// TIA Portal V17 export
// export: Created 2025-03-10T12:14:37.5345526Z, ExportSetting WithDefaults, DisplayName Totally Integrated Automation Portal, DisplayVersion V17 Update 8, DisplayName TIA Portal Openness, DisplayVersion V17 Update 8, DisplayName TIA Portal Version Control Interface, DisplayVersion V17, DisplayName SINAMICS Startdrive Advanced, DisplayVersion V17 SP2, DisplayName SINAMICS Startdrive G110M, G120, G120C, G120D, G120P, G115D, DisplayVersion V17 SP2, DisplayName SINAMICS Startdrive G130, G150, S120, S150, SINAMICS MV, S210, DisplayVersion V17 SP2, DisplayName STEP 7 Professional, DisplayVersion V17 Update 8, DisplayName SINUMERIK ONE STEP 7 Toolbox, DisplayVersion V17 Update 12, DisplayName SINUMERIK 840D sl STEP 7 Toolbox, DisplayVersion V17 Update 12, DisplayName STEP 7 Safety, DisplayVersion V17 Update 6, DisplayName WinCC Advanced, DisplayVersion V17 Update 8
DATA_BLOCK "LBP_SentronPac"   // DB1001
TITLE = for migration: SENTRON PAC / Para migración: SENTRON PAC / für Migration: SENTRON PAC
{ S7_Optimized_Access := 'FALSE'; DB_Accessible_From_OPC_UA := 'FALSE' }
AUTHOR : SINUMERIK
FAMILY : SINUMERIK_ONE
VERSION : 6.15
// for migration: Interface between user program and operating software, contains signals for SENTRON PAC energy monitoring devices / Para migración: interfaz entre programa de usuario y software operativo, contiene señales para dispositivos de control de la energía SENTRON PAC / für Migration: Schnittstelle zwischen Anwenderprogramm und Betriebssoftware, enthält Signale für SENTRON PAC Energieüberwachungsgeräte
// stored: AutoNumber false, DBAccessibleFromOPCUA false, DBAccessibleFromWebserver true, IsOnlyStoredInLoadMemory false, IsWriteProtectedInAS false
   VAR RETAIN
      ManualVal : Bool;   // Anzeige des manuellen Werts / Display of manual value / Indicación del valor manual
      SentronPacMach : Bool;   // Sentron PAC dargestellte Maschine / Sentron PAC represented machine / Máquina representada en Sentron PAC
      FeedInEnergyReadSP : Bool;   // Zugeführte Energie wird von Sentron PAC gelesen / Feed-in energy read from Sentron PAC / La energía suministrada es leída por Sentron PAC
      FeedBackEnergyReadSP : Bool;   // Rückgespeiste Energie wird von Sentron PAC gelesen / Feed back energy read from Sentron PAC / La energía realimentada es leída por Sentron PAC
      FeedInEnergyReadAuxil : Bool;   // Zugeführte Energie, AUX lesen / Feed-in energy read auxiliary / Energía suministrada, leer AUX
      FeedBackEnergyReadAuxil : Bool;   // Rückgespeiste Energie, AUX lesen / Feed back energy read auxiliary / Energía realimentada, leer AUX
      res0_6 : Bool;   // Reserviert / Reserved / Reservado
      res0_7 : Bool;   // Reserviert / Reserved / Reservado
      MeasAuto : Bool;   // Messung durch PLC-Grundprogramm / Measurement by PLC basic program / Medición por programa básico del PLC
      res1_1 : Bool;   // Reserviert / Reserved / Reservado
      res1_2 : Bool;   // Reserviert / Reserved / Reservado
      res1_3 : Bool;   // Reserviert / Reserved / Reservado
      res1_4 : Bool;   // Reserviert / Reserved / Reservado
      res1_5 : Bool;   // Reserviert / Reserved / Reservado
      res1_6 : Bool;   // Reserviert / Reserved / Reservado
      res1_7 : Bool;   // Reserviert / Reserved / Reservado
      MeasAct : Bool;   // Aktive Messung
      res2_1 : Bool;   // Reserviert / Reserved / Reservado
      res2_2 : Bool;   // Reserviert / Reserved / Reservado
      res2_3 : Bool;   // Reserviert / Reserved / Reservado
      res2_4 : Bool;   // Reserviert / Reserved / Reservado
      res2_5 : Bool;   // Reserviert / Reserved / Reservado
      res2_6 : Bool;   // Reserviert / Reserved / Reservado
      res2_7 : Bool;   // Reserviert / Reserved / Reservado
      EStateOn : Bool;   // Energiezustand Ein / Energy state on / Estado energía Con
      res3_1 : Bool;   // Reserviert / Reserved / Reservado
      res3_2 : Bool;   // Reserviert / Reserved / Reservado
      res3_3 : Bool;   // Reserviert / Reserved / Reservado
      res3_4 : Bool;   // Reserviert / Reserved / Reservado
      res3_5 : Bool;   // Reserviert / Reserved / Reservado
      res3_6 : Bool;   // Reserviert / Reserved / Reservado
      res3_7 : Bool;   // Reserviert / Reserved / Reservado
      ManualValue : Real;   // Manueller Wert / Manual value / Valor manual
      ActivePowerItem : Real;   // Wirkleistung Position / Active power item / Potencia activa, posición
      ActiveEnergyItem : Real;   // Wirkenergie Position / Active energy item / Energía activa, posición
      ReactiveEnergyItem : Real;   // Blindenergie Position / Reactive energy item / Energía reactiva, posición
      ActivePowerSentron : Real;   // Wirkleistung von Sentron / Active power from Sentron / Potencia activa de Sentron
      ActiveEnergySentron : Real;   // Wirkenergie von Sentron / Active energy from Sentron / Energía activa de Sentron
      ReactiveEnergySentron : Real;   // Blindenergie von Sentron / Reactive energy from Sentron / Energía reactiva de Sentron
      ActiveEnergyDay : Real;   // Wirkenergie Tag / Active energy day / Energía activa, día
      ReactiveEnergyDay : Real;   // Blindenergie Tag / Reactive energy day / Energía reactiva, día
      ActiveEnergyPrevDay : Real;   // Wirkenergie Vortag / Active energy previous day / Energía activa, día anterior
      ReactiveEnergyPrevDay : Real;   // Blindenergie Vortag / Reactive energy previous day / Energía reactiva, día anterior
      ActiveEnergyMonth : Real;   // Wirkenergie Monat / Active energy month / Energía activa, mes
      ReactiveEnergyMonth : Real;   // Blindenergie Monat / Reactive energy month / Energía reactiva, mes
      ActiveEnergyPrevMonth : Real;   // Wirkenergie Vormonat / Active energy previous month / Energía activa, mes anterior
      ReactiveEnergyPrevMonth : Real;   // Blindenergie Vormonat / Reactive energy previous month / Energía reactiva, mes anterior
      ActiveEnergyYear : Real;   // Wirkenergie Jahr / Active energy year / Energía activa, año
      ReactiveEnergyYear : Real;   // Blindenergie Jahr / Reactive energy year / Energía reactiva, año
      ActiveEnergyPrevYear : Real;   // Wirkenergie Vorjahr / Active energy previous year / Energía activa, año anterior
      ReactiveEnergyPrevYear : Real;   // Blindenergie Vorjahr / Reactive energy previous year / Energía reactiva, año anterior
      res80 : Byte;   // Reserviert / Reserved / Reservado
      res81 : Byte;   // Reserviert / Reserved / Reservado
      res82 : Byte;   // Reserviert / Reserved / Reservado
      res83 : Byte;   // Reserviert / Reserved / Reservado
      res84 : Byte;   // Reserviert / Reserved / Reservado
      res85 : Byte;   // Reserviert / Reserved / Reservado
      res86 : Byte;   // Reserviert / Reserved / Reservado
      res87 : Byte;   // Reserviert / Reserved / Reservado
      res88 : Real;   // Reserviert / Reserved / Reservado
      res92 : Real;   // Reserviert / Reserved / Reservado
      ProductionAct : Byte;
      ErrDBD20_NAN : Bool;   // DBD20: ungültig (keine Nummer) / DBD20: invalid (not a number) / DBD20: no válido (no es número)
      ErrDBD24_NAN : Bool;   // DBD24: ungültig (keine Nummer) / DBD24: invalid (not a number) / DBD24: no válido (no es número)
      ErrDBD28_NAN : Bool;   // DBD28: ungültig (keine Nummer) / DBD28: invalid (not a number) / DBD28: no válido (no es número)
      res97_3 : Bool;   // Reserviert / Reserved / Reservado
      res97_4 : Bool;   // Reserviert / Reserved / Reservado
      res97_5 : Bool;   // Reserviert / Reserved / Reservado
      res97_6 : Bool;   // Reserviert / Reserved / Reservado
      res97_7 : Bool;   // Reserviert / Reserved / Reservado
      ErrDBD104_NAN : Bool;   // DBD104: ungültig (keine Nummer) / DBD104: invalid (not a number) / DBD104: no válido (no es número)
      ErrDBD144_NAN : Bool;   // DBD144: ungültig (keine Nummer) / DBD144: invalid (not a number) / DBD144: no válido (no es número)
      ErrDBD184_NAN : Bool;   // DBD184: ungültig (keine Nummer) / DBD184: invalid (not a number) / DBD184: no válido (no es número)
      ErrDBD224_NAN : Bool;   // DBD224: ungültig (keine Nummer) / DBD224: invalid (not a number) / DBD224: no válido (no es número)
      ErrDBD264_NAN : Bool;   // DBD264: ungültig (keine Nummer) / DBD264: invalid (not a number) / DBD264: no válido (no es número)
      ErrDBD304_NAN : Bool;   // DBD304: ungültig (keine Nummer) / DBD304: invalid (not a number) / DBD304: no válido (no es número)
      ErrDBD344_NAN : Bool;   // DBD344: ungültig (keine Nummer) / DBD344: invalid (not a number) / DBD344: no válido (no es número)
      ErrDBD384_NAN : Bool;   // DBD384: ungültig (keine Nummer) / DBD384: invalid (not a number) / DBD384: no válido (no es número)
      ErrDBD424_NAN : Bool;   // DBD424: ungültig (keine Nummer) / DBD424: invalid (not a number) / DBD424: no válido (no es número)
      ErrDBD464_NAN : Bool;   // DBD464: ungültig (keine Nummer) / DBD464: invalid (not a number) / DBD464: no válido (no es número)
      res99_2 : Bool;   // Reserviert / Reserved / Reservado
      res99_3 : Bool;   // Reserviert / Reserved / Reservado
      res99_4 : Bool;   // Reserviert / Reserved / Reservado
      res99_5 : Bool;   // Reserviert / Reserved / Reservado
      res99_6 : Bool;   // Reserviert / Reserved / Reservado
      res99_7 : Bool;   // Reserviert / Reserved / Reservado
      CtrlE_AuxDevice : Array[1..10] of Struct
         ProcessAux : Bool;   // AUX liegt vor und kann verarbeitet werden / Auxiliary present and to be processed / AUX presente y puede procesarse
         ReadEnergy : Bool;   // Istwerte werden atualisiert; Bit wird automatisch zurückgesetzt / Actual values are refreshed; bit is auto-reset / Los valores reales se actualizan, el bit se resetea automáticamente
         MeasAct : Bool;   // Messwerte werden berechnet / Measurement values are computed / Calculando valores medidos
         MeasMode : Bool;   // Differenz der Istwerte wird gespeichert / Difference of actual values is stored / Guardando diferencia entre valores reales
         InputMode : Bool;   // INPUT "ActivePowerAux" ist Energie in kWh / INPUT "ActivePowerAux" is energy in kWh / INPUT "ActivePowerAux" es energía en kWh
         res0_5 : Bool;
         res0_6 : Bool;
         ResetAux : Bool;   // AUX-Daten werden gelöscht / Auxiliary data are deleted / Los datos AUX se borrarán
         res1 : Byte;   // Reserviert / Reserved / Reservado
         res2 : Word;   // Reserviert / Reserved / Reservado
         ActivePowerAux : Real;   // [kW]/[kWh] Leistung/Energie von AUX, vom Kunden geschrieben / [kW]/[kWh] power/energy of auxiliary, written by customer / [kW]/[kWh] Potencia/energía de AUX, escritas por cliente
         ActiveEnAux : Real;   // [kWh] Istwert der bezogenen Energie / [kWh] actual value of fed-in-energy / [kWh] Valor real de la energía alimentada
         ReActiveEnAux : Real;   // [kWh] Istwert der gelieferten Energie / [kWh] actual value of fed-back energy / [kWh] Valor real de la energía realimentada
         ActiveEnAuxMeasON : Real;   // [kWh] Wert der bezogenen Energie zu Beginn der Messung / [kWh] value of fed-in-energy at start of measurement / [kWh] Valor de la energía alimentada al inicio de la medición
         ReActiveEnAuxMeasON : Real;   // [kWh] Wert der gelieferten Energie zu Beginn der Messung / [kWh] value of fed-back energy at start of measurement / [kWh] Valor de la energía realimentada al inicio de la medición
         ActiveEnAuxMeasOFF : Real;   // [kWh] Wert der bezogenen Energie am Ende der Messung / [kWh] value of fed-in-energy at end of measurement / [kWh] Valor de la energía alimentada al final de la medición
         ReActiveEnAuxMeasOFF : Real;   // [kWh] Wert der gelieferten Energie am Ende der Messung / [kWh] value of fed-back energy at end of measurement / [kWh] Valor de la energía realimentada al final de la medición
         res32 : DWord;   // Reserviert / Reserved / Reservado
         res36 : Real;   // Reserviert / Reserved / Reservado
      END_STRUCT;
   END_VAR
BEGIN
   // CtrlE_AuxDevice[2].ProcessAux : AUX liegt vor und kann verarbeitet werden / Auxiliary present and to be processed / AUX presente y puede procesarse
   // CtrlE_AuxDevice[3].ProcessAux : AUX liegt vor und kann verarbeitet werden / Auxiliary present and to be processed / AUX presente y puede procesarse
   // CtrlE_AuxDevice[4].ProcessAux : AUX liegt vor und kann verarbeitet werden / Auxiliary present and to be processed / AUX presente y puede procesarse
   // CtrlE_AuxDevice[5].ProcessAux : AUX liegt vor und kann verarbeitet werden / Auxiliary present and to be processed / AUX presente y puede procesarse
   // CtrlE_AuxDevice[6].ProcessAux : AUX liegt vor und kann verarbeitet werden / Auxiliary present and to be processed / AUX presente y puede procesarse
   // CtrlE_AuxDevice[7].ProcessAux : AUX liegt vor und kann verarbeitet werden / Auxiliary present and to be processed / AUX presente y puede procesarse
   // CtrlE_AuxDevice[8].ProcessAux : AUX liegt vor und kann verarbeitet werden / Auxiliary present and to be processed / AUX presente y puede procesarse
   // CtrlE_AuxDevice[9].ProcessAux : AUX liegt vor und kann verarbeitet werden / Auxiliary present and to be processed / AUX presente y puede procesarse
   // CtrlE_AuxDevice[10].ProcessAux : AUX liegt vor und kann verarbeitet werden / Auxiliary present and to be processed / AUX presente y puede procesarse
   // CtrlE_AuxDevice[2].ReadEnergy : Istwerte werden atualisiert; Bit wird automatisch zurückgesetzt / Actual values are refreshed; bit is auto-reset / Los valores reales se actualizan, el bit se resetea automáticamente
   // CtrlE_AuxDevice[3].ReadEnergy : Istwerte werden atualisiert; Bit wird automatisch zurückgesetzt / Actual values are refreshed; bit is auto-reset / Los valores reales se actualizan, el bit se resetea automáticamente
   // CtrlE_AuxDevice[4].ReadEnergy : Istwerte werden atualisiert; Bit wird automatisch zurückgesetzt / Actual values are refreshed; bit is auto-reset / Los valores reales se actualizan, el bit se resetea automáticamente
   // CtrlE_AuxDevice[5].ReadEnergy : Istwerte werden atualisiert; Bit wird automatisch zurückgesetzt / Actual values are refreshed; bit is auto-reset / Los valores reales se actualizan, el bit se resetea automáticamente
   // CtrlE_AuxDevice[6].ReadEnergy : Istwerte werden atualisiert; Bit wird automatisch zurückgesetzt / Actual values are refreshed; bit is auto-reset / Los valores reales se actualizan, el bit se resetea automáticamente
   // CtrlE_AuxDevice[7].ReadEnergy : Istwerte werden atualisiert; Bit wird automatisch zurückgesetzt / Actual values are refreshed; bit is auto-reset / Los valores reales se actualizan, el bit se resetea automáticamente
   // CtrlE_AuxDevice[8].ReadEnergy : Istwerte werden atualisiert; Bit wird automatisch zurückgesetzt / Actual values are refreshed; bit is auto-reset / Los valores reales se actualizan, el bit se resetea automáticamente
   // CtrlE_AuxDevice[9].ReadEnergy : Istwerte werden atualisiert; Bit wird automatisch zurückgesetzt / Actual values are refreshed; bit is auto-reset / Los valores reales se actualizan, el bit se resetea automáticamente
   // CtrlE_AuxDevice[10].ReadEnergy : Istwerte werden atualisiert; Bit wird automatisch zurückgesetzt / Actual values are refreshed; bit is auto-reset / Los valores reales se actualizan, el bit se resetea automáticamente
   // CtrlE_AuxDevice[2].MeasAct : Messwerte werden berechnet / Measurement values are computed / Calculando valores medidos
   // CtrlE_AuxDevice[3].MeasAct : Messwerte werden berechnet / Measurement values are computed / Calculando valores medidos
   // CtrlE_AuxDevice[4].MeasAct : Messwerte werden berechnet / Measurement values are computed / Calculando valores medidos
   // CtrlE_AuxDevice[5].MeasAct : Messwerte werden berechnet / Measurement values are computed / Calculando valores medidos
   // CtrlE_AuxDevice[6].MeasAct : Messwerte werden berechnet / Measurement values are computed / Calculando valores medidos
   // CtrlE_AuxDevice[7].MeasAct : Messwerte werden berechnet / Measurement values are computed / Calculando valores medidos
   // CtrlE_AuxDevice[8].MeasAct : Messwerte werden berechnet / Measurement values are computed / Calculando valores medidos
   // CtrlE_AuxDevice[9].MeasAct : Messwerte werden berechnet / Measurement values are computed / Calculando valores medidos
   // CtrlE_AuxDevice[10].MeasAct : Messwerte werden berechnet / Measurement values are computed / Calculando valores medidos
   // CtrlE_AuxDevice[2].MeasMode : Differenz der Istwerte wird gespeichert / Difference of actual values is stored / Guardando diferencia entre valores reales
   // CtrlE_AuxDevice[3].MeasMode : Differenz der Istwerte wird gespeichert / Difference of actual values is stored / Guardando diferencia entre valores reales
   // CtrlE_AuxDevice[4].MeasMode : Differenz der Istwerte wird gespeichert / Difference of actual values is stored / Guardando diferencia entre valores reales
   // CtrlE_AuxDevice[5].MeasMode : Differenz der Istwerte wird gespeichert / Difference of actual values is stored / Guardando diferencia entre valores reales
   // CtrlE_AuxDevice[6].MeasMode : Differenz der Istwerte wird gespeichert / Difference of actual values is stored / Guardando diferencia entre valores reales
   // CtrlE_AuxDevice[7].MeasMode : Differenz der Istwerte wird gespeichert / Difference of actual values is stored / Guardando diferencia entre valores reales
   // CtrlE_AuxDevice[8].MeasMode : Differenz der Istwerte wird gespeichert / Difference of actual values is stored / Guardando diferencia entre valores reales
   // CtrlE_AuxDevice[9].MeasMode : Differenz der Istwerte wird gespeichert / Difference of actual values is stored / Guardando diferencia entre valores reales
   // CtrlE_AuxDevice[10].MeasMode : Differenz der Istwerte wird gespeichert / Difference of actual values is stored / Guardando diferencia entre valores reales
   // CtrlE_AuxDevice[2].InputMode : INPUT "ActivePowerAux" ist Energie in kWh / INPUT "ActivePowerAux" is energy in kWh / INPUT "ActivePowerAux" es energía en kWh
   // CtrlE_AuxDevice[3].InputMode : INPUT "ActivePowerAux" ist Energie in kWh / INPUT "ActivePowerAux" is energy in kWh / INPUT "ActivePowerAux" es energía en kWh
   // CtrlE_AuxDevice[4].InputMode : INPUT "ActivePowerAux" ist Energie in kWh / INPUT "ActivePowerAux" is energy in kWh / INPUT "ActivePowerAux" es energía en kWh
   // CtrlE_AuxDevice[5].InputMode : INPUT "ActivePowerAux" ist Energie in kWh / INPUT "ActivePowerAux" is energy in kWh / INPUT "ActivePowerAux" es energía en kWh
   // CtrlE_AuxDevice[6].InputMode : INPUT "ActivePowerAux" ist Energie in kWh / INPUT "ActivePowerAux" is energy in kWh / INPUT "ActivePowerAux" es energía en kWh
   // CtrlE_AuxDevice[7].InputMode : INPUT "ActivePowerAux" ist Energie in kWh / INPUT "ActivePowerAux" is energy in kWh / INPUT "ActivePowerAux" es energía en kWh
   // CtrlE_AuxDevice[8].InputMode : INPUT "ActivePowerAux" ist Energie in kWh / INPUT "ActivePowerAux" is energy in kWh / INPUT "ActivePowerAux" es energía en kWh
   // CtrlE_AuxDevice[9].InputMode : INPUT "ActivePowerAux" ist Energie in kWh / INPUT "ActivePowerAux" is energy in kWh / INPUT "ActivePowerAux" es energía en kWh
   // CtrlE_AuxDevice[10].InputMode : INPUT "ActivePowerAux" ist Energie in kWh / INPUT "ActivePowerAux" is energy in kWh / INPUT "ActivePowerAux" es energía en kWh
   // CtrlE_AuxDevice[2].ResetAux : AUX-Daten werden gelöscht / Auxiliary data are deleted / Los datos AUX se borrarán
   // CtrlE_AuxDevice[3].ResetAux : AUX-Daten werden gelöscht / Auxiliary data are deleted / Los datos AUX se borrarán
   // CtrlE_AuxDevice[4].ResetAux : AUX-Daten werden gelöscht / Auxiliary data are deleted / Los datos AUX se borrarán
   // CtrlE_AuxDevice[5].ResetAux : AUX-Daten werden gelöscht / Auxiliary data are deleted / Los datos AUX se borrarán
   // CtrlE_AuxDevice[6].ResetAux : AUX-Daten werden gelöscht / Auxiliary data are deleted / Los datos AUX se borrarán
   // CtrlE_AuxDevice[7].ResetAux : AUX-Daten werden gelöscht / Auxiliary data are deleted / Los datos AUX se borrarán
   // CtrlE_AuxDevice[8].ResetAux : AUX-Daten werden gelöscht / Auxiliary data are deleted / Los datos AUX se borrarán
   // CtrlE_AuxDevice[9].ResetAux : AUX-Daten werden gelöscht / Auxiliary data are deleted / Los datos AUX se borrarán
   // CtrlE_AuxDevice[10].ResetAux : AUX-Daten werden gelöscht / Auxiliary data are deleted / Los datos AUX se borrarán
   // CtrlE_AuxDevice[2].res1 : Reserviert / Reserved / Reservado
   // CtrlE_AuxDevice[3].res1 : Reserviert / Reserved / Reservado
   // CtrlE_AuxDevice[4].res1 : Reserviert / Reserved / Reservado
   // CtrlE_AuxDevice[5].res1 : Reserviert / Reserved / Reservado
   // CtrlE_AuxDevice[6].res1 : Reserviert / Reserved / Reservado
   // CtrlE_AuxDevice[7].res1 : Reserviert / Reserved / Reservado
   // CtrlE_AuxDevice[8].res1 : Reserviert / Reserved / Reservado
   // CtrlE_AuxDevice[9].res1 : Reserviert / Reserved / Reservado
   // CtrlE_AuxDevice[10].res1 : Reserviert / Reserved / Reservado
   // CtrlE_AuxDevice[2].res2 : Reserviert / Reserved / Reservado
   // CtrlE_AuxDevice[3].res2 : Reserviert / Reserved / Reservado
   // CtrlE_AuxDevice[4].res2 : Reserviert / Reserved / Reservado
   // CtrlE_AuxDevice[5].res2 : Reserviert / Reserved / Reservado
   // CtrlE_AuxDevice[6].res2 : Reserviert / Reserved / Reservado
   // CtrlE_AuxDevice[7].res2 : Reserviert / Reserved / Reservado
   // CtrlE_AuxDevice[8].res2 : Reserviert / Reserved / Reservado
   // CtrlE_AuxDevice[9].res2 : Reserviert / Reserved / Reservado
   // CtrlE_AuxDevice[10].res2 : Reserviert / Reserved / Reservado
   // CtrlE_AuxDevice[2].ActivePowerAux : [kW]/[kWh] Leistung/Energie von AUX, vom Kunden geschrieben / [kW]/[kWh] power/energy of auxiliary, written by customer / [kW]/[kWh] Potencia/energía de AUX, escritas por cliente
   // CtrlE_AuxDevice[3].ActivePowerAux : [kW]/[kWh] Leistung/Energie von AUX, vom Kunden geschrieben / [kW]/[kWh] power/energy of auxiliary, written by customer / [kW]/[kWh] Potencia/energía de AUX, escritas por cliente
   // CtrlE_AuxDevice[4].ActivePowerAux : [kW]/[kWh] Leistung/Energie von AUX, vom Kunden geschrieben / [kW]/[kWh] power/energy of auxiliary, written by customer / [kW]/[kWh] Potencia/energía de AUX, escritas por cliente
   // CtrlE_AuxDevice[5].ActivePowerAux : [kW]/[kWh] Leistung/Energie von AUX, vom Kunden geschrieben / [kW]/[kWh] power/energy of auxiliary, written by customer / [kW]/[kWh] Potencia/energía de AUX, escritas por cliente
   // CtrlE_AuxDevice[6].ActivePowerAux : [kW]/[kWh] Leistung/Energie von AUX, vom Kunden geschrieben / [kW]/[kWh] power/energy of auxiliary, written by customer / [kW]/[kWh] Potencia/energía de AUX, escritas por cliente
   // CtrlE_AuxDevice[7].ActivePowerAux : [kW]/[kWh] Leistung/Energie von AUX, vom Kunden geschrieben / [kW]/[kWh] power/energy of auxiliary, written by customer / [kW]/[kWh] Potencia/energía de AUX, escritas por cliente
   // CtrlE_AuxDevice[8].ActivePowerAux : [kW]/[kWh] Leistung/Energie von AUX, vom Kunden geschrieben / [kW]/[kWh] power/energy of auxiliary, written by customer / [kW]/[kWh] Potencia/energía de AUX, escritas por cliente
   // CtrlE_AuxDevice[9].ActivePowerAux : [kW]/[kWh] Leistung/Energie von AUX, vom Kunden geschrieben / [kW]/[kWh] power/energy of auxiliary, written by customer / [kW]/[kWh] Potencia/energía de AUX, escritas por cliente
   // CtrlE_AuxDevice[10].ActivePowerAux : [kW]/[kWh] Leistung/Energie von AUX, vom Kunden geschrieben / [kW]/[kWh] power/energy of auxiliary, written by customer / [kW]/[kWh] Potencia/energía de AUX, escritas por cliente
   // CtrlE_AuxDevice[2].ActiveEnAux : [kWh] Istwert der bezogenen Energie / [kWh] actual value of fed-in-energy / [kWh] Valor real de la energía alimentada
   // CtrlE_AuxDevice[3].ActiveEnAux : [kWh] Istwert der bezogenen Energie / [kWh] actual value of fed-in-energy / [kWh] Valor real de la energía alimentada
   // CtrlE_AuxDevice[4].ActiveEnAux : [kWh] Istwert der bezogenen Energie / [kWh] actual value of fed-in-energy / [kWh] Valor real de la energía alimentada
   // CtrlE_AuxDevice[5].ActiveEnAux : [kWh] Istwert der bezogenen Energie / [kWh] actual value of fed-in-energy / [kWh] Valor real de la energía alimentada
   // CtrlE_AuxDevice[6].ActiveEnAux : [kWh] Istwert der bezogenen Energie / [kWh] actual value of fed-in-energy / [kWh] Valor real de la energía alimentada
   // CtrlE_AuxDevice[7].ActiveEnAux : [kWh] Istwert der bezogenen Energie / [kWh] actual value of fed-in-energy / [kWh] Valor real de la energía alimentada
   // CtrlE_AuxDevice[8].ActiveEnAux : [kWh] Istwert der bezogenen Energie / [kWh] actual value of fed-in-energy / [kWh] Valor real de la energía alimentada
   // CtrlE_AuxDevice[9].ActiveEnAux : [kWh] Istwert der bezogenen Energie / [kWh] actual value of fed-in-energy / [kWh] Valor real de la energía alimentada
   // CtrlE_AuxDevice[10].ActiveEnAux : [kWh] Istwert der bezogenen Energie / [kWh] actual value of fed-in-energy / [kWh] Valor real de la energía alimentada
   // CtrlE_AuxDevice[2].ReActiveEnAux : [kWh] Istwert der gelieferten Energie / [kWh] actual value of fed-back energy / [kWh] Valor real de la energía realimentada
   // CtrlE_AuxDevice[3].ReActiveEnAux : [kWh] Istwert der gelieferten Energie / [kWh] actual value of fed-back energy / [kWh] Valor real de la energía realimentada
   // CtrlE_AuxDevice[4].ReActiveEnAux : [kWh] Istwert der gelieferten Energie / [kWh] actual value of fed-back energy / [kWh] Valor real de la energía realimentada
   // CtrlE_AuxDevice[5].ReActiveEnAux : [kWh] Istwert der gelieferten Energie / [kWh] actual value of fed-back energy / [kWh] Valor real de la energía realimentada
   // CtrlE_AuxDevice[6].ReActiveEnAux : [kWh] Istwert der gelieferten Energie / [kWh] actual value of fed-back energy / [kWh] Valor real de la energía realimentada
   // CtrlE_AuxDevice[7].ReActiveEnAux : [kWh] Istwert der gelieferten Energie / [kWh] actual value of fed-back energy / [kWh] Valor real de la energía realimentada
   // CtrlE_AuxDevice[8].ReActiveEnAux : [kWh] Istwert der gelieferten Energie / [kWh] actual value of fed-back energy / [kWh] Valor real de la energía realimentada
   // CtrlE_AuxDevice[9].ReActiveEnAux : [kWh] Istwert der gelieferten Energie / [kWh] actual value of fed-back energy / [kWh] Valor real de la energía realimentada
   // CtrlE_AuxDevice[10].ReActiveEnAux : [kWh] Istwert der gelieferten Energie / [kWh] actual value of fed-back energy / [kWh] Valor real de la energía realimentada
   // CtrlE_AuxDevice[2].ActiveEnAuxMeasON : [kWh] Wert der bezogenen Energie zu Beginn der Messung / [kWh] value of fed-in-energy at start of measurement / [kWh] Valor de la energía alimentada al inicio de la medición
   // CtrlE_AuxDevice[3].ActiveEnAuxMeasON : [kWh] Wert der bezogenen Energie zu Beginn der Messung / [kWh] value of fed-in-energy at start of measurement / [kWh] Valor de la energía alimentada al inicio de la medición
   // CtrlE_AuxDevice[4].ActiveEnAuxMeasON : [kWh] Wert der bezogenen Energie zu Beginn der Messung / [kWh] value of fed-in-energy at start of measurement / [kWh] Valor de la energía alimentada al inicio de la medición
   // CtrlE_AuxDevice[5].ActiveEnAuxMeasON : [kWh] Wert der bezogenen Energie zu Beginn der Messung / [kWh] value of fed-in-energy at start of measurement / [kWh] Valor de la energía alimentada al inicio de la medición
   // CtrlE_AuxDevice[6].ActiveEnAuxMeasON : [kWh] Wert der bezogenen Energie zu Beginn der Messung / [kWh] value of fed-in-energy at start of measurement / [kWh] Valor de la energía alimentada al inicio de la medición
   // CtrlE_AuxDevice[7].ActiveEnAuxMeasON : [kWh] Wert der bezogenen Energie zu Beginn der Messung / [kWh] value of fed-in-energy at start of measurement / [kWh] Valor de la energía alimentada al inicio de la medición
   // CtrlE_AuxDevice[8].ActiveEnAuxMeasON : [kWh] Wert der bezogenen Energie zu Beginn der Messung / [kWh] value of fed-in-energy at start of measurement / [kWh] Valor de la energía alimentada al inicio de la medición
   // CtrlE_AuxDevice[9].ActiveEnAuxMeasON : [kWh] Wert der bezogenen Energie zu Beginn der Messung / [kWh] value of fed-in-energy at start of measurement / [kWh] Valor de la energía alimentada al inicio de la medición
   // CtrlE_AuxDevice[10].ActiveEnAuxMeasON : [kWh] Wert der bezogenen Energie zu Beginn der Messung / [kWh] value of fed-in-energy at start of measurement / [kWh] Valor de la energía alimentada al inicio de la medición
   // CtrlE_AuxDevice[2].ReActiveEnAuxMeasON : [kWh] Wert der gelieferten Energie zu Beginn der Messung / [kWh] value of fed-back energy at start of measurement / [kWh] Valor de la energía realimentada al inicio de la medición
   // CtrlE_AuxDevice[3].ReActiveEnAuxMeasON : [kWh] Wert der gelieferten Energie zu Beginn der Messung / [kWh] value of fed-back energy at start of measurement / [kWh] Valor de la energía realimentada al inicio de la medición
   // CtrlE_AuxDevice[4].ReActiveEnAuxMeasON : [kWh] Wert der gelieferten Energie zu Beginn der Messung / [kWh] value of fed-back energy at start of measurement / [kWh] Valor de la energía realimentada al inicio de la medición
   // CtrlE_AuxDevice[5].ReActiveEnAuxMeasON : [kWh] Wert der gelieferten Energie zu Beginn der Messung / [kWh] value of fed-back energy at start of measurement / [kWh] Valor de la energía realimentada al inicio de la medición
   // CtrlE_AuxDevice[6].ReActiveEnAuxMeasON : [kWh] Wert der gelieferten Energie zu Beginn der Messung / [kWh] value of fed-back energy at start of measurement / [kWh] Valor de la energía realimentada al inicio de la medición
   // CtrlE_AuxDevice[7].ReActiveEnAuxMeasON : [kWh] Wert der gelieferten Energie zu Beginn der Messung / [kWh] value of fed-back energy at start of measurement / [kWh] Valor de la energía realimentada al inicio de la medición
   // CtrlE_AuxDevice[8].ReActiveEnAuxMeasON : [kWh] Wert der gelieferten Energie zu Beginn der Messung / [kWh] value of fed-back energy at start of measurement / [kWh] Valor de la energía realimentada al inicio de la medición
   // CtrlE_AuxDevice[9].ReActiveEnAuxMeasON : [kWh] Wert der gelieferten Energie zu Beginn der Messung / [kWh] value of fed-back energy at start of measurement / [kWh] Valor de la energía realimentada al inicio de la medición
   // CtrlE_AuxDevice[10].ReActiveEnAuxMeasON : [kWh] Wert der gelieferten Energie zu Beginn der Messung / [kWh] value of fed-back energy at start of measurement / [kWh] Valor de la energía realimentada al inicio de la medición
   // CtrlE_AuxDevice[2].ActiveEnAuxMeasOFF : [kWh] Wert der bezogenen Energie am Ende der Messung / [kWh] value of fed-in-energy at end of measurement / [kWh] Valor de la energía alimentada al final de la medición
   // CtrlE_AuxDevice[3].ActiveEnAuxMeasOFF : [kWh] Wert der bezogenen Energie am Ende der Messung / [kWh] value of fed-in-energy at end of measurement / [kWh] Valor de la energía alimentada al final de la medición
   // CtrlE_AuxDevice[4].ActiveEnAuxMeasOFF : [kWh] Wert der bezogenen Energie am Ende der Messung / [kWh] value of fed-in-energy at end of measurement / [kWh] Valor de la energía alimentada al final de la medición
   // CtrlE_AuxDevice[5].ActiveEnAuxMeasOFF : [kWh] Wert der bezogenen Energie am Ende der Messung / [kWh] value of fed-in-energy at end of measurement / [kWh] Valor de la energía alimentada al final de la medición
   // CtrlE_AuxDevice[6].ActiveEnAuxMeasOFF : [kWh] Wert der bezogenen Energie am Ende der Messung / [kWh] value of fed-in-energy at end of measurement / [kWh] Valor de la energía alimentada al final de la medición
   // CtrlE_AuxDevice[7].ActiveEnAuxMeasOFF : [kWh] Wert der bezogenen Energie am Ende der Messung / [kWh] value of fed-in-energy at end of measurement / [kWh] Valor de la energía alimentada al final de la medición
   // CtrlE_AuxDevice[8].ActiveEnAuxMeasOFF : [kWh] Wert der bezogenen Energie am Ende der Messung / [kWh] value of fed-in-energy at end of measurement / [kWh] Valor de la energía alimentada al final de la medición
   // CtrlE_AuxDevice[9].ActiveEnAuxMeasOFF : [kWh] Wert der bezogenen Energie am Ende der Messung / [kWh] value of fed-in-energy at end of measurement / [kWh] Valor de la energía alimentada al final de la medición
   // CtrlE_AuxDevice[10].ActiveEnAuxMeasOFF : [kWh] Wert der bezogenen Energie am Ende der Messung / [kWh] value of fed-in-energy at end of measurement / [kWh] Valor de la energía alimentada al final de la medición
   // CtrlE_AuxDevice[2].ReActiveEnAuxMeasOFF : [kWh] Wert der gelieferten Energie am Ende der Messung / [kWh] value of fed-back energy at end of measurement / [kWh] Valor de la energía realimentada al final de la medición
   // CtrlE_AuxDevice[3].ReActiveEnAuxMeasOFF : [kWh] Wert der gelieferten Energie am Ende der Messung / [kWh] value of fed-back energy at end of measurement / [kWh] Valor de la energía realimentada al final de la medición
   // CtrlE_AuxDevice[4].ReActiveEnAuxMeasOFF : [kWh] Wert der gelieferten Energie am Ende der Messung / [kWh] value of fed-back energy at end of measurement / [kWh] Valor de la energía realimentada al final de la medición
   // CtrlE_AuxDevice[5].ReActiveEnAuxMeasOFF : [kWh] Wert der gelieferten Energie am Ende der Messung / [kWh] value of fed-back energy at end of measurement / [kWh] Valor de la energía realimentada al final de la medición
   // CtrlE_AuxDevice[6].ReActiveEnAuxMeasOFF : [kWh] Wert der gelieferten Energie am Ende der Messung / [kWh] value of fed-back energy at end of measurement / [kWh] Valor de la energía realimentada al final de la medición
   // CtrlE_AuxDevice[7].ReActiveEnAuxMeasOFF : [kWh] Wert der gelieferten Energie am Ende der Messung / [kWh] value of fed-back energy at end of measurement / [kWh] Valor de la energía realimentada al final de la medición
   // CtrlE_AuxDevice[8].ReActiveEnAuxMeasOFF : [kWh] Wert der gelieferten Energie am Ende der Messung / [kWh] value of fed-back energy at end of measurement / [kWh] Valor de la energía realimentada al final de la medición
   // CtrlE_AuxDevice[9].ReActiveEnAuxMeasOFF : [kWh] Wert der gelieferten Energie am Ende der Messung / [kWh] value of fed-back energy at end of measurement / [kWh] Valor de la energía realimentada al final de la medición
   // CtrlE_AuxDevice[10].ReActiveEnAuxMeasOFF : [kWh] Wert der gelieferten Energie am Ende der Messung / [kWh] value of fed-back energy at end of measurement / [kWh] Valor de la energía realimentada al final de la medición
   // CtrlE_AuxDevice[2].res32 : Reserviert / Reserved / Reservado
   // CtrlE_AuxDevice[3].res32 : Reserviert / Reserved / Reservado
   // CtrlE_AuxDevice[4].res32 : Reserviert / Reserved / Reservado
   // CtrlE_AuxDevice[5].res32 : Reserviert / Reserved / Reservado
   // CtrlE_AuxDevice[6].res32 : Reserviert / Reserved / Reservado
   // CtrlE_AuxDevice[7].res32 : Reserviert / Reserved / Reservado
   // CtrlE_AuxDevice[8].res32 : Reserviert / Reserved / Reservado
   // CtrlE_AuxDevice[9].res32 : Reserviert / Reserved / Reservado
   // CtrlE_AuxDevice[10].res32 : Reserviert / Reserved / Reservado
   // CtrlE_AuxDevice[2].res36 : Reserviert / Reserved / Reservado
   // CtrlE_AuxDevice[3].res36 : Reserviert / Reserved / Reservado
   // CtrlE_AuxDevice[4].res36 : Reserviert / Reserved / Reservado
   // CtrlE_AuxDevice[5].res36 : Reserviert / Reserved / Reservado
   // CtrlE_AuxDevice[6].res36 : Reserviert / Reserved / Reservado
   // CtrlE_AuxDevice[7].res36 : Reserviert / Reserved / Reservado
   // CtrlE_AuxDevice[8].res36 : Reserviert / Reserved / Reservado
   // CtrlE_AuxDevice[9].res36 : Reserviert / Reserved / Reservado
   // CtrlE_AuxDevice[10].res36 : Reserviert / Reserved / Reservado
END_DATA_BLOCK
